// TIA Portal project "analog input test" (V14)

(* hardware
DEVICE "S7-1200 station_1"  S7-1200 Station
   slot 0: "Rack_0"  S7-1200 Rack  Rack  V1.0
   slot 1: "PLC_1"  CPU 1214C DC/DC/DC  6ES7 214-1AG40-0XB0  V4.2
   slot 2: "AI 4x13BIT_1"  6ES7 231-4HD32-0XB0  V2.0
   slot 3: "AI 4x13BIT_2"  6ES7 231-4HD32-0XB0  V2.0
   slot 4: "AI 4xTC_1"  SM 1231 AI4 x TC  6ES7 231-5QD32-0XB0  V2.0
   slot 5: "AI 4xTC_2"  SM 1231 AI4 x TC  6ES7 231-5QD32-0XB0  V2.0
   slot 6: "AI 4xTC_3"  SM 1231 AI4 x TC  6ES7 231-5QD32-0XB0  V2.0
   slot 101: "CM 1241 (RS422/485)_1"  6ES7 241-1CH32-0XB0  V2.2
*)

// ===== PLC "PLC_1"  CPU 1214C DC/DC/DC =====

VAR_GLOBAL   // PLC tag table "Default tag table"
   "Analog Input 1" AT %IW64 : Int;
   "Analog Input 2" AT %IW66 : Int;
   "Pressure Transducer 1" AT %IW96 : Int;
   "Pressure Transducer 2" AT %IW98 : Int;
   "Pressure Transducer 3" AT %IW100 : Int;
   "Pressure Transducer 4" AT %IW102 : Int;
   "Pressure Transducer 5" AT %IW112 : Int;
   "Pressure Transducer 6" AT %IW114 : Int;
   "Pressure Transducer 7" AT %IW116 : Int;
   "Pressure Transducer 8" AT %IW118 : Int;
   "Thermocouple 1" AT %IW128 : Word;
   "Thermocouple 2" AT %IW130 : Word;
   "Thermocouple 3" AT %IW132 : Word;
   "Thermocouple 4" AT %IW134 : Word;
   "Thermocouple 5" AT %IW144 : Word;
   "Thermocouple 6" AT %IW146 : Word;
   "Thermocouple 7" AT %IW148 : Word;
   "Thermocouple 8" AT %IW150 : Word;
   "Thermocouple 9" AT %IW160 : Word;
   "Thermocouple 10" AT %IW162 : Word;
   "Thermocouple 11" AT %IW164 : Word;
   "Thermocouple 12" AT %IW166 : Word;
   "Boolean Test" AT %M1000.0 : Bool;
   "Test" AT %M1000.1 : Bool;
   "Tag_1" AT %I0.4 : Bool;
END_VAR

DATA_BLOCK "Data_block_1"   // DB1
{ S7_Optimized_Access := 'TRUE' }
VERSION : 0.1
   VAR
      "Int Test" : Int;
   END_VAR
BEGIN
END_DATA_BLOCK

DATA_BLOCK "MB Holding Reg"   // DB2
{ S7_Optimized_Access := 'TRUE' }
VERSION : 0.1
   VAR
      MB40k : Array[1..100] of Word;
   END_VAR
BEGIN
   // MB40k[1] : Pressure Transducer 1
   // MB40k[2] : Pressure Transducer 2
   // MB40k[3] : Pressure 3
   // MB40k[4] : Pressure 4
   // MB40k[5] : Pressure 5
   // MB40k[6] : Pressure 6
   // MB40k[7] : Pressure 7
   // MB40k[8] : Pressure 8
   // MB40k[9] : Tempurature 1
   // MB40k[10] : Tempurature 2
   // MB40k[11] : Tempuratere 3
   // MB40k[12] : Temp4
   // MB40k[13] : temp 5
   // MB40k[14] : temp6
   // MB40k[15] : temp7
   // MB40k[16] : temp8
   // MB40k[17] : temp9
   // MB40k[18] : temp10
   // MB40k[19] : temp11
   // MB40k[20] : temp12
END_DATA_BLOCK

DATA_BLOCK "Normalize Temporary Values"   // DB3
{ S7_Optimized_Access := 'TRUE' }
VERSION : 0.1
   VAR
      "Pressure Norm Temp 1" : Real;
      "Pressure Norm Temp 2" : Real;
      "Pressure Norm Temp 3" : Real;
      "Pressure Norm Temp 4" : Real;
      "Pressure Norm Temp 5" : Real;
      "Pressure Norm Temp 6" : Real;
      "Pressure Norm Temp 7" : Real;
      "Pressure Norm Temp 8" : Real;
   END_VAR
BEGIN
END_DATA_BLOCK

DATA_BLOCK "Data_block_4"   // DB5
{ S7_Optimized_Access := 'TRUE' }
VERSION : 0.1
   VAR
      "Static 1" : Real;
      "Static 2" : Real;
      "kpa 1" : Real;
      "Psi 1" : Word;
   END_VAR
BEGIN
END_DATA_BLOCK

DATA_BLOCK "Modbus communication"   // DB7
{ S7_Optimized_Access := 'TRUE' }
VERSION : 0.1
   VAR
      Comms : TCON_IP_v4;
   END_VAR
BEGIN
   Comms.InterfaceId := 64;
   Comms.ID := 1;
   Comms.RemoteAddress.ADDR[1] := 192;
   Comms.RemoteAddress.ADDR[2] := 168;
   Comms.RemoteAddress.ADDR[3] := 1;
   Comms.RemoteAddress.ADDR[4] := 13;
   Comms.LocalPort := 502;
END_DATA_BLOCK

FUNCTION_BLOCK "Convert Pressure Input to kpa"   // FB1, LAD
{ S7_Optimized_Access := 'TRUE' }
VERSION : 0.1
   VAR_INPUT
      "Analog Input" : Int;
      "Raw input at -7kpa" : Int;
      "Raw input at 7kpa" : Int;
   END_VAR
   VAR_OUTPUT
      kpa : Real;
   END_VAR
   VAR_TEMP
      "Normed Value" : Real;
   END_VAR
BEGIN

REGION Network 2
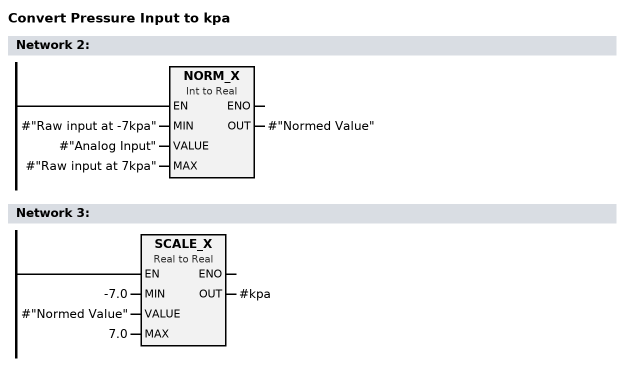
   RUNG wire#powerrail
      { S7_Templates := "[SrcType := Int, DestType := Real]" } Normalize(min := #"Raw input at -7kpa", value := #"Analog Input", max := #"Raw input at 7kpa", out => #"Normed Value")
   END_RUNG
   // the same network as SCL:
   #"Normed Value" := NORM_X(MIN := #"Raw input at -7kpa", VALUE := #"Analog Input", MAX := #"Raw input at 7kpa");
END_REGION

REGION Network 3
   RUNG wire#powerrail
      { S7_Templates := "[SrcType := Real, DestType := Real]" } Scale(min := -7.0, value := #"Normed Value", max := 7.0, out => #kpa)
   END_RUNG
   // the same network as SCL:
   #kpa := SCALE_X(MIN := -7.0, VALUE := #"Normed Value", MAX := 7.0);
END_REGION
END_FUNCTION_BLOCK

FUNCTION "Conevert Pressure input to PSI" : Void   // FC1, LAD
{ S7_Optimized_Access := 'TRUE' }
VERSION : 0.1
   VAR_INPUT
      "Raw input at 0psi" : Real;
      "Raw input at 1psi" : Real;
      "Analog input address" : Real;
   END_VAR
   VAR_OUTPUT
      Psi : Real;
   END_VAR
   VAR_TEMP
      "Raw input at -1 psi" : Real;
      "Psi Math" : Real;
      "Normalized Value" : Real;
      "real psi" : Real;
   END_VAR
BEGIN

REGION Network 1
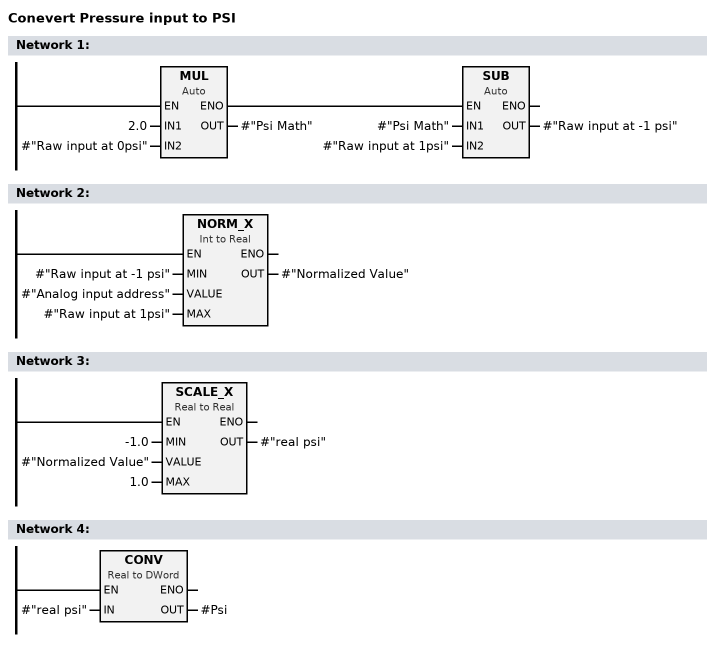
   RUNG wire#powerrail
      Mul(in1 := 2.0, in2 := #"Raw input at 0psi", out => #"Psi Math")
      Sub(in1 := #"Psi Math", in2 := #"Raw input at 1psi", out => #"Raw input at -1 psi")
   END_RUNG
   // the same network as SCL:
   #"Psi Math" := 2.0 * #"Raw input at 0psi";
   #"Raw input at -1 psi" := #"Psi Math" - #"Raw input at 1psi";
END_REGION

REGION Network 2
   RUNG wire#powerrail
      { S7_Templates := "[SrcType := Int, DestType := Real]" } Normalize(min := #"Raw input at -1 psi", value := #"Analog input address", max := #"Raw input at 1psi", out => #"Normalized Value")
   END_RUNG
   // the same network as SCL:
   #"Normalized Value" := NORM_X(MIN := #"Raw input at -1 psi", VALUE := #"Analog input address", MAX := #"Raw input at 1psi");
END_REGION

REGION Network 3
   RUNG wire#powerrail
      { S7_Templates := "[SrcType := Real, DestType := Real]" } Scale(min := -1.0, value := #"Normalized Value", max := 1.0, out => #"real psi")
   END_RUNG
   // the same network as SCL:
   #"real psi" := SCALE_X(MIN := -1.0, VALUE := #"Normalized Value", MAX := 1.0);
END_REGION

REGION Network 4
   RUNG wire#powerrail
      { S7_Templates := "[SrcType := Real, DestType := DWord]" } Convert(in := #"real psi", out => #Psi)
   END_RUNG
   // the same network as SCL:
   #Psi := REAL_TO_DWORD(#"real psi");
END_REGION
END_FUNCTION

ORGANIZATION_BLOCK "Main"   // OB1, LAD, ProgramCycle
TITLE = "Main Program Sweep (Cycle)"
{ S7_Optimized_Access := 'TRUE' }
VERSION : 0.1
   VAR_INPUT
      Initial_Call : Bool;   // Initial call of this OB
      Remanence : Bool;   // =True, if remanent data are available
   END_VAR
BEGIN

REGION Network 1: Setup Mos
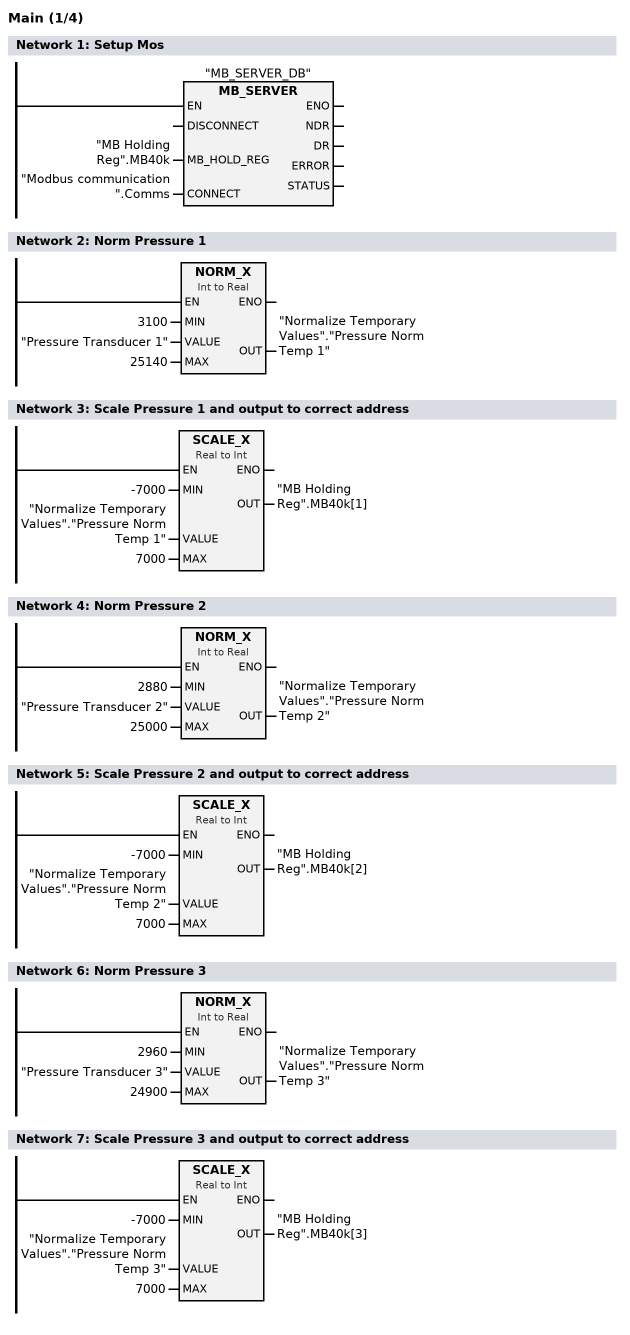
   "MB_SERVER_DB"(MB_HOLD_REG := "MB Holding Reg".MB40k, CONNECT := "Modbus communication".Comms);   // MB_SERVER
END_REGION

REGION Network 2: Norm Pressure 1
   RUNG wire#powerrail
      { S7_Templates := "[SrcType := Int, DestType := Real]" } Normalize(min := 3100, value := "Pressure Transducer 1", max := 25140, out => "Normalize Temporary Values"."Pressure Norm Temp 1")
   END_RUNG
   // the same network as SCL:
   "Normalize Temporary Values"."Pressure Norm Temp 1" := NORM_X(MIN := 3100, VALUE := "Pressure Transducer 1", MAX := 25140);
END_REGION

REGION Network 3: Scale Pressure 1 and output to correct address
   RUNG wire#powerrail
      { S7_Templates := "[SrcType := Real, DestType := Int]" } Scale(min := -7000, value := "Normalize Temporary Values"."Pressure Norm Temp 1", max := 7000, out => "MB Holding Reg".MB40k[1])
   END_RUNG
   // the same network as SCL:
   "MB Holding Reg".MB40k[1] := SCALE_X(MIN := -7000, VALUE := "Normalize Temporary Values"."Pressure Norm Temp 1", MAX := 7000);
END_REGION

REGION Network 4: Norm Pressure 2
   RUNG wire#powerrail
      { S7_Templates := "[SrcType := Int, DestType := Real]" } Normalize(min := 2880, value := "Pressure Transducer 2", max := 25000, out => "Normalize Temporary Values"."Pressure Norm Temp 2")
   END_RUNG
   // the same network as SCL:
   "Normalize Temporary Values"."Pressure Norm Temp 2" := NORM_X(MIN := 2880, VALUE := "Pressure Transducer 2", MAX := 25000);
END_REGION

REGION Network 5: Scale Pressure 2 and output to correct address
   RUNG wire#powerrail
      { S7_Templates := "[SrcType := Real, DestType := Int]" } Scale(min := -7000, value := "Normalize Temporary Values"."Pressure Norm Temp 2", max := 7000, out => "MB Holding Reg".MB40k[2])
   END_RUNG
   // the same network as SCL:
   "MB Holding Reg".MB40k[2] := SCALE_X(MIN := -7000, VALUE := "Normalize Temporary Values"."Pressure Norm Temp 2", MAX := 7000);
END_REGION

REGION Network 6: Norm Pressure 3
   RUNG wire#powerrail
      { S7_Templates := "[SrcType := Int, DestType := Real]" } Normalize(min := 2960, value := "Pressure Transducer 3", max := 24900, out => "Normalize Temporary Values"."Pressure Norm Temp 3")
   END_RUNG
   // the same network as SCL:
   "Normalize Temporary Values"."Pressure Norm Temp 3" := NORM_X(MIN := 2960, VALUE := "Pressure Transducer 3", MAX := 24900);
END_REGION

REGION Network 7: Scale Pressure 3 and output to correct address
   RUNG wire#powerrail
      { S7_Templates := "[SrcType := Real, DestType := Int]" } Scale(min := -7000, value := "Normalize Temporary Values"."Pressure Norm Temp 3", max := 7000, out => "MB Holding Reg".MB40k[3])
   END_RUNG
   // the same network as SCL:
   "MB Holding Reg".MB40k[3] := SCALE_X(MIN := -7000, VALUE := "Normalize Temporary Values"."Pressure Norm Temp 3", MAX := 7000);
END_REGION

REGION Network 8: Norm Pressure 4
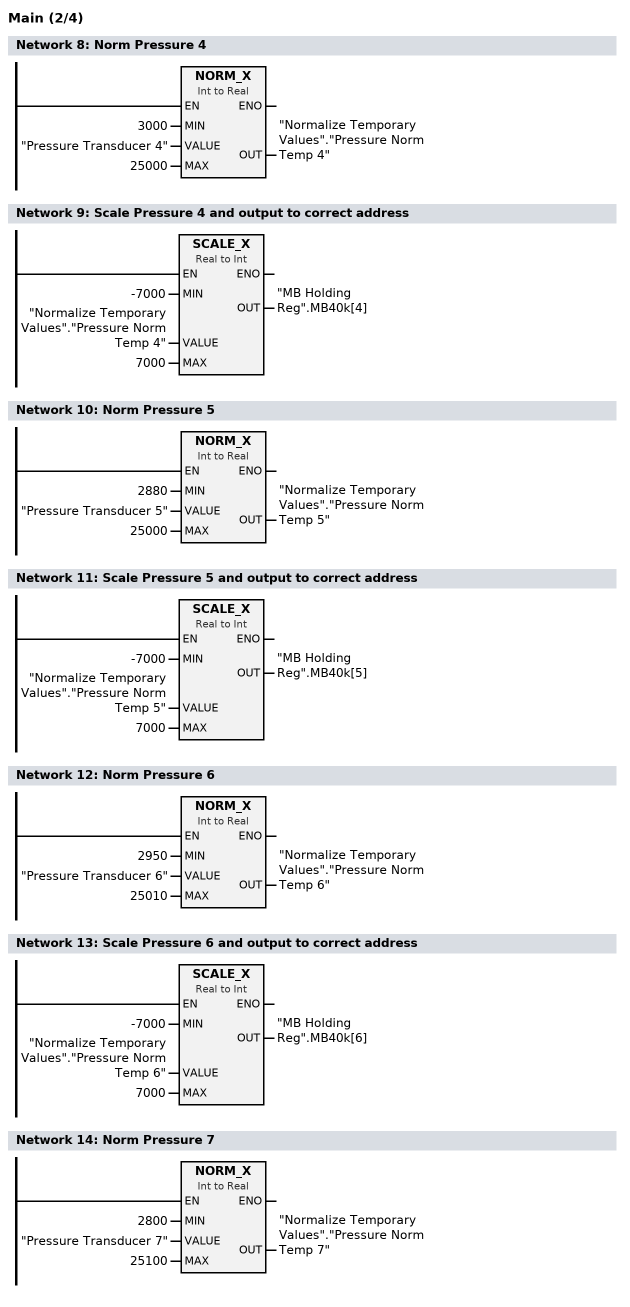
   RUNG wire#powerrail
      { S7_Templates := "[SrcType := Int, DestType := Real]" } Normalize(min := 3000, value := "Pressure Transducer 4", max := 25000, out => "Normalize Temporary Values"."Pressure Norm Temp 4")
   END_RUNG
   // the same network as SCL:
   "Normalize Temporary Values"."Pressure Norm Temp 4" := NORM_X(MIN := 3000, VALUE := "Pressure Transducer 4", MAX := 25000);
END_REGION

REGION Network 9: Scale Pressure 4 and output to correct address
   RUNG wire#powerrail
      { S7_Templates := "[SrcType := Real, DestType := Int]" } Scale(min := -7000, value := "Normalize Temporary Values"."Pressure Norm Temp 4", max := 7000, out => "MB Holding Reg".MB40k[4])
   END_RUNG
   // the same network as SCL:
   "MB Holding Reg".MB40k[4] := SCALE_X(MIN := -7000, VALUE := "Normalize Temporary Values"."Pressure Norm Temp 4", MAX := 7000);
END_REGION

REGION Network 10: Norm Pressure 5
   RUNG wire#powerrail
      { S7_Templates := "[SrcType := Int, DestType := Real]" } Normalize(min := 2880, value := "Pressure Transducer 5", max := 25000, out => "Normalize Temporary Values"."Pressure Norm Temp 5")
   END_RUNG
   // the same network as SCL:
   "Normalize Temporary Values"."Pressure Norm Temp 5" := NORM_X(MIN := 2880, VALUE := "Pressure Transducer 5", MAX := 25000);
END_REGION

REGION Network 11: Scale Pressure 5 and output to correct address
   RUNG wire#powerrail
      { S7_Templates := "[SrcType := Real, DestType := Int]" } Scale(min := -7000, value := "Normalize Temporary Values"."Pressure Norm Temp 5", max := 7000, out => "MB Holding Reg".MB40k[5])
   END_RUNG
   // the same network as SCL:
   "MB Holding Reg".MB40k[5] := SCALE_X(MIN := -7000, VALUE := "Normalize Temporary Values"."Pressure Norm Temp 5", MAX := 7000);
END_REGION

REGION Network 12: Norm Pressure 6
   RUNG wire#powerrail
      { S7_Templates := "[SrcType := Int, DestType := Real]" } Normalize(min := 2950, value := "Pressure Transducer 6", max := 25010, out => "Normalize Temporary Values"."Pressure Norm Temp 6")
   END_RUNG
   // the same network as SCL:
   "Normalize Temporary Values"."Pressure Norm Temp 6" := NORM_X(MIN := 2950, VALUE := "Pressure Transducer 6", MAX := 25010);
END_REGION

REGION Network 13: Scale Pressure 6 and output to correct address
   RUNG wire#powerrail
      { S7_Templates := "[SrcType := Real, DestType := Int]" } Scale(min := -7000, value := "Normalize Temporary Values"."Pressure Norm Temp 6", max := 7000, out => "MB Holding Reg".MB40k[6])
   END_RUNG
   // the same network as SCL:
   "MB Holding Reg".MB40k[6] := SCALE_X(MIN := -7000, VALUE := "Normalize Temporary Values"."Pressure Norm Temp 6", MAX := 7000);
END_REGION

REGION Network 14: Norm Pressure 7
   RUNG wire#powerrail
      { S7_Templates := "[SrcType := Int, DestType := Real]" } Normalize(min := 2800, value := "Pressure Transducer 7", max := 25100, out => "Normalize Temporary Values"."Pressure Norm Temp 7")
   END_RUNG
   // the same network as SCL:
   "Normalize Temporary Values"."Pressure Norm Temp 7" := NORM_X(MIN := 2800, VALUE := "Pressure Transducer 7", MAX := 25100);
END_REGION

REGION Network 15: Scale Pressure 7 and output to correct address
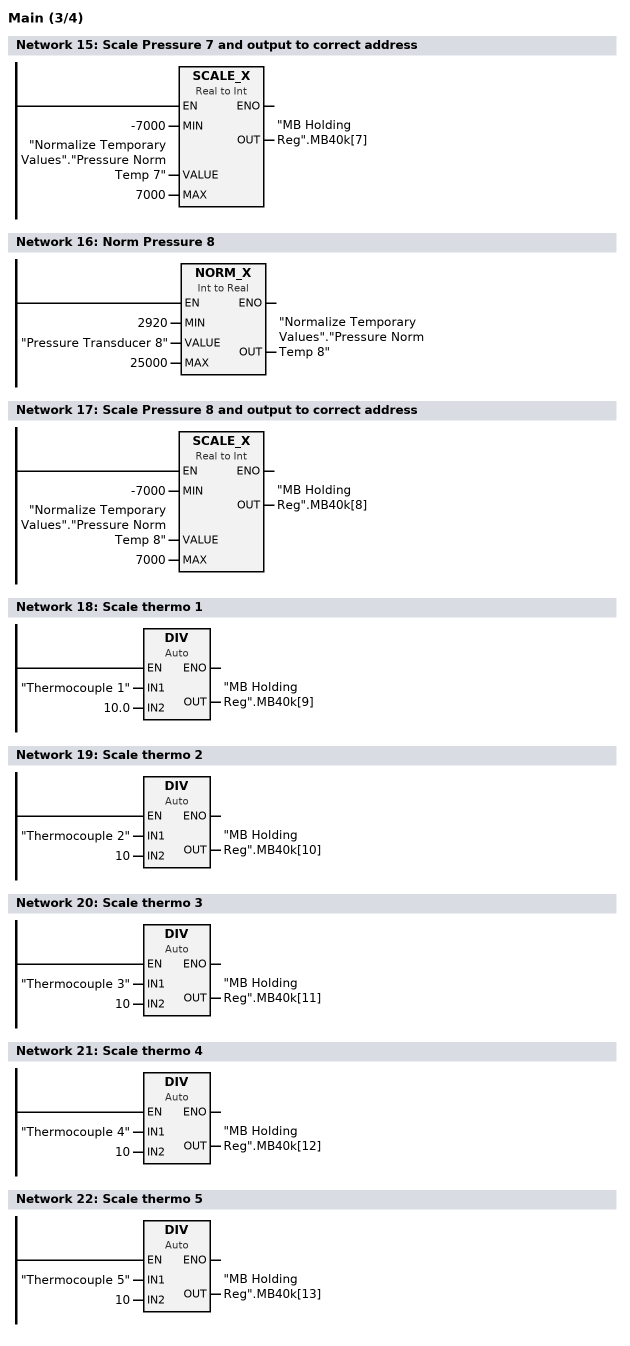
   RUNG wire#powerrail
      { S7_Templates := "[SrcType := Real, DestType := Int]" } Scale(min := -7000, value := "Normalize Temporary Values"."Pressure Norm Temp 7", max := 7000, out => "MB Holding Reg".MB40k[7])
   END_RUNG
   // the same network as SCL:
   "MB Holding Reg".MB40k[7] := SCALE_X(MIN := -7000, VALUE := "Normalize Temporary Values"."Pressure Norm Temp 7", MAX := 7000);
END_REGION

REGION Network 16: Norm Pressure 8
   RUNG wire#powerrail
      { S7_Templates := "[SrcType := Int, DestType := Real]" } Normalize(min := 2920, value := "Pressure Transducer 8", max := 25000, out => "Normalize Temporary Values"."Pressure Norm Temp 8")
   END_RUNG
   // the same network as SCL:
   "Normalize Temporary Values"."Pressure Norm Temp 8" := NORM_X(MIN := 2920, VALUE := "Pressure Transducer 8", MAX := 25000);
END_REGION

REGION Network 17: Scale Pressure 8 and output to correct address
   RUNG wire#powerrail
      { S7_Templates := "[SrcType := Real, DestType := Int]" } Scale(min := -7000, value := "Normalize Temporary Values"."Pressure Norm Temp 8", max := 7000, out => "MB Holding Reg".MB40k[8])
   END_RUNG
   // the same network as SCL:
   "MB Holding Reg".MB40k[8] := SCALE_X(MIN := -7000, VALUE := "Normalize Temporary Values"."Pressure Norm Temp 8", MAX := 7000);
END_REGION

REGION Network 18: Scale thermo 1
   RUNG wire#powerrail
      Div(in1 := "Thermocouple 1", in2 := 10.0, out => "MB Holding Reg".MB40k[9])
   END_RUNG
   // the same network as SCL:
   "MB Holding Reg".MB40k[9] := "Thermocouple 1" / 10.0;
END_REGION

REGION Network 19: Scale thermo 2
   RUNG wire#powerrail
      Div(in1 := "Thermocouple 2", in2 := 10, out => "MB Holding Reg".MB40k[10])
   END_RUNG
   // the same network as SCL:
   "MB Holding Reg".MB40k[10] := "Thermocouple 2" / 10;
END_REGION

REGION Network 20: Scale thermo 3
   RUNG wire#powerrail
      Div(in1 := "Thermocouple 3", in2 := 10, out => "MB Holding Reg".MB40k[11])
   END_RUNG
   // the same network as SCL:
   "MB Holding Reg".MB40k[11] := "Thermocouple 3" / 10;
END_REGION

REGION Network 21: Scale thermo 4
   RUNG wire#powerrail
      Div(in1 := "Thermocouple 4", in2 := 10, out => "MB Holding Reg".MB40k[12])
   END_RUNG
   // the same network as SCL:
   "MB Holding Reg".MB40k[12] := "Thermocouple 4" / 10;
END_REGION

REGION Network 22: Scale thermo 5
   RUNG wire#powerrail
      Div(in1 := "Thermocouple 5", in2 := 10, out => "MB Holding Reg".MB40k[13])
   END_RUNG
   // the same network as SCL:
   "MB Holding Reg".MB40k[13] := "Thermocouple 5" / 10;
END_REGION

REGION Network 23: Scale thermo 6
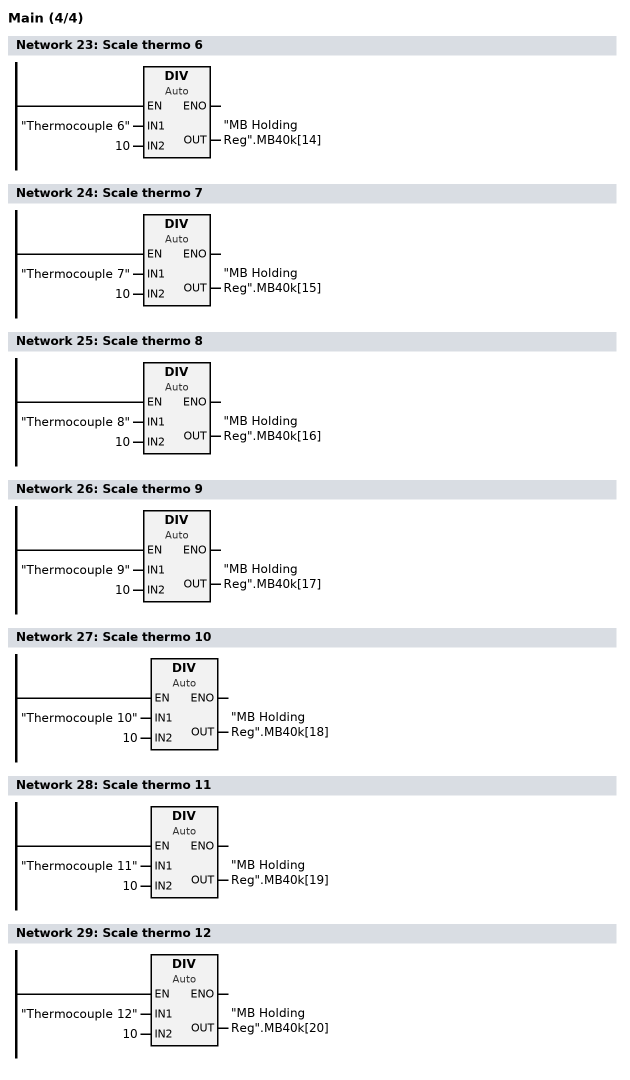
   RUNG wire#powerrail
      Div(in1 := "Thermocouple 6", in2 := 10, out => "MB Holding Reg".MB40k[14])
   END_RUNG
   // the same network as SCL:
   "MB Holding Reg".MB40k[14] := "Thermocouple 6" / 10;
END_REGION

REGION Network 24: Scale thermo 7
   RUNG wire#powerrail
      Div(in1 := "Thermocouple 7", in2 := 10, out => "MB Holding Reg".MB40k[15])
   END_RUNG
   // the same network as SCL:
   "MB Holding Reg".MB40k[15] := "Thermocouple 7" / 10;
END_REGION

REGION Network 25: Scale thermo 8
   RUNG wire#powerrail
      Div(in1 := "Thermocouple 8", in2 := 10, out => "MB Holding Reg".MB40k[16])
   END_RUNG
   // the same network as SCL:
   "MB Holding Reg".MB40k[16] := "Thermocouple 8" / 10;
END_REGION

REGION Network 26: Scale thermo 9
   RUNG wire#powerrail
      Div(in1 := "Thermocouple 9", in2 := 10, out => "MB Holding Reg".MB40k[17])
   END_RUNG
   // the same network as SCL:
   "MB Holding Reg".MB40k[17] := "Thermocouple 9" / 10;
END_REGION

REGION Network 27: Scale thermo 10
   RUNG wire#powerrail
      Div(in1 := "Thermocouple 10", in2 := 10, out => "MB Holding Reg".MB40k[18])
   END_RUNG
   // the same network as SCL:
   "MB Holding Reg".MB40k[18] := "Thermocouple 10" / 10;
END_REGION

REGION Network 28: Scale thermo 11
   RUNG wire#powerrail
      Div(in1 := "Thermocouple 11", in2 := 10, out => "MB Holding Reg".MB40k[19])
   END_RUNG
   // the same network as SCL:
   "MB Holding Reg".MB40k[19] := "Thermocouple 11" / 10;
END_REGION

REGION Network 29: Scale thermo 12
   RUNG wire#powerrail
      Div(in1 := "Thermocouple 12", in2 := 10, out => "MB Holding Reg".MB40k[20])
   END_RUNG
   // the same network as SCL:
   "MB Holding Reg".MB40k[20] := "Thermocouple 12" / 10;
END_REGION
END_ORGANIZATION_BLOCK